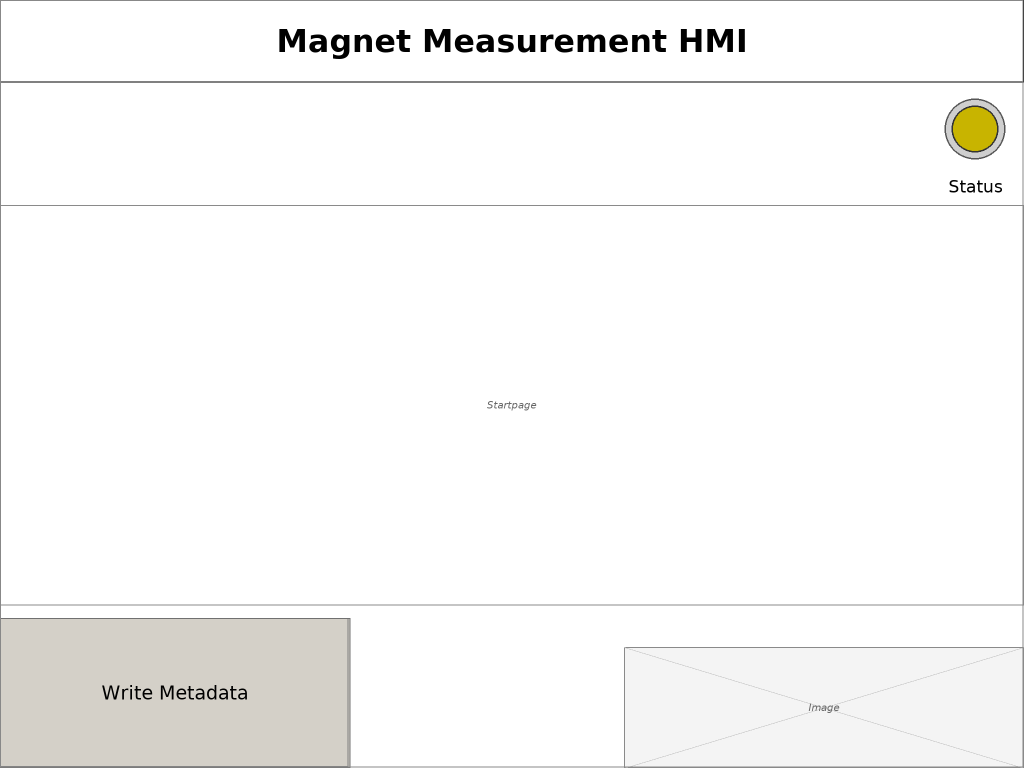
VISUALIZATION Visualization  // 1024x768
    Button (0,618 350x150), "Write Metadata"
        OnMouseClick: FrameSelectionChange Selection=SelectedFrame=f10d8547-6667-49de-9f33-336b6c15e565, Selection=1, GlobSel=AssignType=Directly, SelType=Locally
    RoundedRectangle (0,0 1024x82), "Magnet Measurement HMI"
    Image (624,647 400x121)
        p84334746: 'BAM_Logo'
    Lamp1 (940,94 70x70), tooltip "Status", style: Lamp-Lamp1-Yellow
    Label (941,167 70x39), "Status"
    Frame (0,205 1024x400)
        shows Startpage()
        shows Write_Metadata_Visu()
END_VISUALIZATION

(* stored: Version 1.1.0.1, ProductVersion 3.1.4024.12
   Visu Visualization: Id {16194027-daab-4e64-8353-062eb5c814c0} *)
